// User API for interlocks, add each new interlocks interface here
INTERFACE I_MotionInterlocks

METHOD AxisStatus
VAR_INPUT
	HomeBusy: BOOL;
	PositiveDirection : BOOL;
	NegativeDirection : BOOL;
END_VAR
END_METHOD

METHOD DriveCommands
VAR_INPUT
	Enable: BOOL;
	NewMoveReq : BOOL;
END_VAR
END_METHOD

PROPERTY Error : BOOL
GET
END_GET
END_PROPERTY

PROPERTY ErrorID : UDINT
GET
END_GET
END_PROPERTY

PROPERTY InterlockEvent : BOOL
GET
END_GET
END_PROPERTY

PROPERTY LimHome : BOOL
GET
END_GET
END_PROPERTY

PROPERTY Message : T_MAXSTRING
GET
END_GET
END_PROPERTY

PROPERTY MoveBackwardEnabled : BOOL
GET
END_GET
END_PROPERTY

PROPERTY MoveForwardEnabled : BOOL
GET
END_GET
END_PROPERTY

PROPERTY MoveOk : BOOL
GET
END_GET
END_PROPERTY

PROPERTY PowerEnabled : BOOL
GET
END_GET
END_PROPERTY

METHOD Reset
VAR_INPUT
END_VAR
END_METHOD

PROPERTY Warning : BOOL
GET
END_GET
END_PROPERTY

END_INTERFACE

(* stored: Version 1.1.0.1
   Itf I_MotionInterlocks: Id {f1e8e58f-70bb-485c-99bb-95a56820fdb6}
   Method AxisStatus: Id {dacb7d42-f913-4c3c-8725-5ac4315a091a}
   Method DriveCommands: Id {4eadfef4-5c7c-464f-b3d8-85555ae4b8ba}
   Property Error: Id {cb8c4f4f-26d3-4070-a3b0-01084a7b31fd}
   Get Get: Id {3c954f64-0417-4db1-abeb-dec4d46a007d}
   Property ErrorID: Id {3679fc85-f898-430b-b18e-92a8643354fe}
   Get Get: Id {f7bc3532-00ad-4cf2-8f15-5d20c5cbe6d9}
   Property InterlockEvent: Id {4626fde1-1a12-4e8c-af56-a81a21e2e625}
   Get Get: Id {46f4e7d2-165f-43e2-b11a-41b0ae0b097d}
   Property LimHome: Id {afb29fce-e002-4581-b44c-7cdfce3976d7}
   Get Get: Id {c5ce7826-2bcf-4ef7-a3c3-f2af2474caae}
   Property Message: Id {9f0d5caf-5e8b-49a6-9cb6-a74ac978daca}
   Get Get: Id {5e7d9b57-4a23-4d1a-ae3d-a3c1e73b4ad0}
   Property MoveBackwardEnabled: Id {437d5026-d3d2-451f-aaec-a79f11811b76}
   Get Get: Id {7c34fb6f-f131-4c32-8007-32b5760134e0}
   Property MoveForwardEnabled: Id {3f0479ef-0797-4b11-80d8-e2af512406d5}
   Get Get: Id {c48ed286-fb7c-46b5-b434-3eb5c4175687}
   Property MoveOk: Id {923a20cb-b75b-46f9-bb2a-200129f48beb}
   Get Get: Id {0ff386a4-7805-4634-a7c9-b25a0c9fccc6}
   Property PowerEnabled: Id {21374bb6-d388-4443-be9e-3f9b640d7d98}
   Get Get: Id {84d4d810-7c5b-4fb1-848b-e406f6d15e58}
   Method Reset: Id {5eaf8c93-8e83-434e-8bc9-866213c3ec76}
   Property Warning: Id {91e00cec-1c9c-45a9-adce-d11447c803e6}
   Get Get: Id {24c57123-3d83-4dfc-8d6f-96a327d66a69} *)
